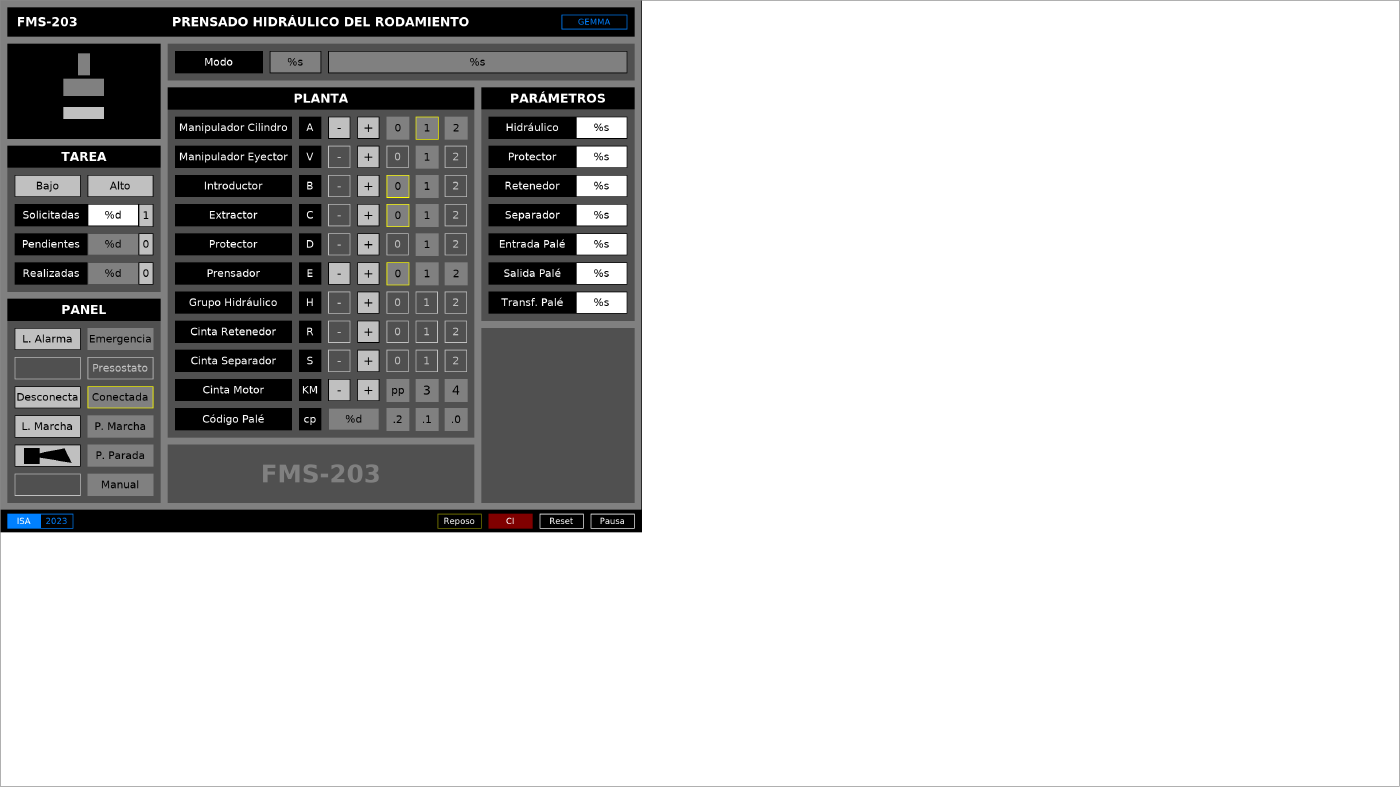
VISUALIZATION TC_VISU  // 1920x1080
    Rectangle (120,610 90x30)
    Rectangle (0,0 880x700)
    Rectangle (230,150 420x450)
    Rectangle (10,440 210x250)
    Rectangle (10,10 860x40), "PRENSADO HIDRÁULICO DEL RODAMIENTO"
    Rectangle (770,20 90x20), "GEMMA"
    Rectangle (10,60 210x130)
    Rectangle (230,120 420x30), "PLANTA"
    Rectangle (240,160 160x30), "Manipulador Cilindro"
    Rectangle (410,160 30x30), "A"
    Rectangle (450,160 30x30), "-"
    Rectangle (490,160 30x30), "+"
    Rectangle (530,160 30x30), "0"
    Rectangle (570,160 30x30), "1"
    Rectangle (610,160 30x30), "2"
    Rectangle (530,160 31x31), "0", colour toggle: MAIN.Estacion.ManipuladorDetras
        toggle MAIN.Estacion.ManipuladorDetras
    Rectangle (490,160 30x30), "+", colour toggle: MAIN.Estacion.ManipuladorAdelante
        toggle MAIN.Estacion.ManipuladorAdelante
    Rectangle (570,160 31x31), "1", colour toggle: MAIN.Estacion.ManipuladorMedio
        toggle MAIN.Estacion.ManipuladorMedio
    Rectangle (240,240 160x30), "Introductor"
    Rectangle (410,240 30x30), "B"
    Rectangle (10,410 210x30), "PANEL"
    Rectangle (20,450 90x30)
    Rectangle (0,700 880x30)
    Rectangle (55,705 45x20), "2023"
    Rectangle (10,705 45x20), "ISA"
    Rectangle (20,490 90x30)
    Rectangle (120,490 90x30), "Presostato"
    Rectangle (20,530 90x30)
    Rectangle (20,570 90x30)
    Rectangle (20,610 90x30)
    Rectangle (20,650 90x30)
    Rectangle (20,450 90x30), "L. Alarma", colour toggle: MAIN.Estacion.LamparaAlarma
        tap MAIN.Estacion.LamparaAlarma
    Rectangle (20,530 90x30), "Desconecta", colour toggle: MAIN.Estacion.DesconectaEstacion
        tap MAIN.Estacion.DesconectaEstacion
    Rectangle (20,570 90x30), "L. Marcha", colour toggle: MAIN.Estacion.LamparaMarcha
        tap MAIN.Estacion.LamparaMarcha
    Rectangle (20,610 90x30), colour toggle: MAIN.Estacion.AvisadorSonoro
        tap MAIN.Estacion.AvisadorSonoro
    Rectangle (120,450 90x30), colour toggle: MAIN.Estacion.PulsadorEmergencia
        toggle MAIN.Estacion.PulsadorEmergencia
    Rectangle (120,570 90x30)
    Rectangle (120,530 90x30)
    Rectangle (120,650 90x30)
    Rectangle (240,280 160x30), "Extractor"
    Rectangle (410,280 30x30), "C"
    Rectangle (240,320 160x30), "Protector"
    Rectangle (410,320 30x30), "D"
    Rectangle (240,360 160x30), "Prensador"
    Rectangle (410,360 30x30), "E"
    Rectangle (240,200 160x30), "Manipulador Eyector"
    Rectangle (410,200 30x30), "V"
    Rectangle (240,400 160x30), "Grupo Hidráulico"
    Rectangle (410,400 30x30), "H"
    Rectangle (240,440 160x30), "Cinta Retenedor"
    Rectangle (410,440 30x30), "R"
    Rectangle (240,480 160x30), "Cinta Separador"
    Rectangle (410,480 30x30), "S"
    Rectangle (240,520 160x30), "Cinta Motor"
    Rectangle (410,520 30x30), "KM"
    Rectangle (240,560 160x30), "Código Palé"
    Rectangle (410,560 30x30), "cp"
    Rectangle (230,610 420x80), "FMS-203"
    Rectangle (450,240 30x30), "-"
    Rectangle (490,240 30x30), "+"
    Rectangle (530,240 30x30), "0"
    Rectangle (570,240 30x30), "1"
    Rectangle (610,240 30x30), "2"
    Rectangle (530,240 31x31), "0", colour toggle: MAIN.Estacion.IntroductorDetras
        toggle MAIN.Estacion.IntroductorDetras
    Rectangle (490,240 30x30), "+", colour toggle: MAIN.Estacion.IntroductorAdelante
        toggle MAIN.Estacion.IntroductorAdelante
    Rectangle (570,240 31x31), "1", colour toggle: MAIN.Estacion.IntroductorDelante
        toggle MAIN.Estacion.IntroductorDelante
    Rectangle (450,280 30x30), "-"
    Rectangle (490,280 30x30), "+"
    Rectangle (530,280 30x30), "0"
    Rectangle (570,280 30x30), "1"
    Rectangle (610,280 30x30), "2"
    Rectangle (530,280 31x31), "0", colour toggle: MAIN.Estacion.ExtractorDetras
        toggle MAIN.Estacion.ExtractorDetras
    Rectangle (490,280 30x30), "+", colour toggle: MAIN.Estacion.ExtractorAdelante
        toggle MAIN.Estacion.ExtractorAdelante
    Rectangle (570,280 31x31), "1", colour toggle: MAIN.Estacion.ExtractorDelante
        toggle MAIN.Estacion.ExtractorDelante
    Rectangle (450,320 30x30), "-"
    Rectangle (490,320 30x30), "+"
    Rectangle (530,320 30x30), "0"
    Rectangle (570,320 30x30), "1"
    Rectangle (610,320 30x30), "2"
    Rectangle (490,320 30x30), "+", colour toggle: MAIN.Estacion.ProtectorBaja
        toggle MAIN.Estacion.ProtectorBaja
    Rectangle (570,320 31x31), "1", colour toggle: MAIN.Estacion.ProtectorAbajo
        toggle MAIN.Estacion.ProtectorAbajo
    Rectangle (450,360 30x30), "-"
    Rectangle (490,360 30x30), "+"
    Rectangle (530,360 30x30), "0"
    Rectangle (570,360 30x30), "1"
    Rectangle (610,360 30x30), "2"
    Rectangle (530,360 31x31), "0", colour toggle: MAIN.Estacion.PrensadorArriba
        toggle MAIN.Estacion.PrensadorArriba
    Rectangle (490,360 30x30), "+", colour toggle: MAIN.Estacion.PrensadorBaja
        toggle MAIN.Estacion.PrensadorBaja
    Rectangle (570,360 31x31), "1", colour toggle: MAIN.Estacion.PrensadorAbajoAlto
        toggle MAIN.Estacion.PrensadorAbajoAlto
    Rectangle (610,360 31x31), "2", colour toggle: MAIN.Estacion.PrensadorAbajoBajo
        toggle MAIN.Estacion.PrensadorAbajoBajo
    Rectangle (450,200 30x30), "-"
    Rectangle (450,360 30x30), "-", colour toggle: MAIN.Estacion.PrensadorSube
        toggle MAIN.Estacion.PrensadorSube
    Rectangle (490,200 30x30), "+"
    Rectangle (530,200 30x30), "0"
    Rectangle (570,200 30x30), "1"
    Rectangle (610,200 30x30), "2"
    Rectangle (490,200 30x30), "+", colour toggle: MAIN.Estacion.ManipuladorSucciona
        toggle MAIN.Estacion.ManipuladorSucciona
    Rectangle (570,200 31x31), "1", colour toggle: MAIN.Estacion.ManipuladorVacioObtenido
        toggle MAIN.Estacion.ManipuladorVacioObtenido
    Rectangle (450,400 30x30), "-"
    Rectangle (490,400 30x30), "+"
    Rectangle (530,400 30x30), "0"
    Rectangle (570,400 30x30), "1"
    Rectangle (610,400 30x30), "2"
    Rectangle (490,400 30x30), "+", colour toggle: MAIN.Estacion.HidraulicoActiva
        toggle MAIN.Estacion.HidraulicoActiva
    Rectangle (450,440 30x30), "-"
    Rectangle (490,440 30x30), "+"
    Rectangle (530,440 30x30), "0"
    Rectangle (570,440 30x30), "1"
    Rectangle (610,440 30x30), "2"
    Rectangle (490,440 30x30), "+", colour toggle: MAIN.Estacion.CintaRetenedorBaja
        toggle MAIN.Estacion.CintaRetenedorBaja
    Rectangle (450,480 30x30), "-"
    Rectangle (490,480 30x30), "+"
    Rectangle (530,480 30x30), "0"
    Rectangle (570,480 30x30), "1"
    Rectangle (610,480 30x30), "2"
    Rectangle (490,480 30x30), "+", colour toggle: MAIN.Estacion.CintaSeparadorSube
        toggle MAIN.Estacion.CintaSeparadorSube
    Rectangle (450,520 30x30), "-"
    Rectangle (450,520 30x30), "-", colour toggle: MAIN.Estacion.CintaMotorInvierte
        toggle MAIN.Estacion.CintaMotorInvierte
    Rectangle (490,520 30x30), "+"
    Rectangle (530,520 30x30), "0"
    Rectangle (570,520 30x30), "1"
    Rectangle (610,520 30x30), "2"
    Rectangle (530,520 31x31), "pp", colour toggle: MAIN.Estacion.PalePresencia
        toggle MAIN.Estacion.PalePresencia
    Rectangle (490,520 30x30), "+", colour toggle: MAIN.Estacion.CintaMotorActiva
        toggle MAIN.Estacion.CintaMotorActiva
    Rectangle (570,520 31x31), "3", colour toggle: MAIN.Estacion.CintaMotorActiva AND MAIN.Estacion.CintaMotorInvierte
    Rectangle (450,560 30x30), "-"
    Rectangle (490,560 30x30), "+"
    Rectangle (530,560 30x30), "0"
    Rectangle (570,560 30x30), "1"
    Rectangle (610,560 30x30), "2"
    Rectangle (530,560 31x31), ".2", colour toggle: MAIN.Estacion.PaleCodigoBit2
        toggle MAIN.Estacion.PaleCodigoBit2
    Rectangle (610,560 31x31), ".0", colour toggle: MAIN.Estacion.PaleCodigoBit0
        toggle MAIN.Estacion.PaleCodigoBit0
    Rectangle (570,560 31x31), ".1", colour toggle: MAIN.Estacion.PaleCodigoBit1
        toggle MAIN.Estacion.PaleCodigoBit1
    Rectangle (450,560 70x30), "%d", text variable: MAIN.Estacion.PaleCodigo
    Rectangle (610,520 31x31), "4", colour toggle: MAIN.Estacion.CintaMotorActiva AND NOT MAIN.Estacion.CintaMotorInvierte
    Rectangle (120,530 90x30), "Conectada", colour toggle: MAIN.Estacion.EstacionConectada
        toggle MAIN.Estacion.EstacionConectada
    Rectangle (120,570 90x30), "P. Marcha", colour toggle: MAIN.Estacion.PulsadorMarcha
        tap MAIN.Estacion.PulsadorMarcha
    Rectangle (120,450 90x30), "Emergencia", colour toggle: MAIN.Estacion.PulsadorEmergencia
        toggle MAIN.Estacion.PulsadorEmergencia
    Rectangle (120,650 90x30), "Manual", colour toggle: MAIN.Estacion.SelectorManual
        toggle MAIN.Estacion.SelectorManual
    Rectangle (120,610 90x30)
    Rectangle (120,610 90x30), "P. Parada", colour toggle: MAIN.Estacion.PulsadorParada
        tap MAIN.Estacion.PulsadorParada p1329445385=TRUE
    Group (56,71 119x109)
        Group (0,0 117x107)
            Polygon (119,109)
            Polygon (0,109)
            Polyline (40,94)
            Polyline (30,86)
            Polyline (30,76)
            Polyline (30,66)
            Polyline (40,54)
            Polyline (119,104)
            Polyline (119,94)
            Polyline (119,84)
            Polyline (119,74)
            Polyline (119,54)
            Rectangle (29,35 59x27)
            Rectangle (49,0 20x34)
            Rectangle (49,22 20x12)
            Rectangle (29,63 59x10)
            Polyline (40,104)
            Polyline (118,64)
            Rectangle (29,74 59x20)
        Polygon (119,109)
        Polygon (0,109)
        Polyline (40,94)
        Polyline (30,86)
        Polyline (30,76)
        Polyline (30,66)
        Polyline (40,54)
        Polyline (119,104)
        Polyline (119,94)
        Polyline (119,84)
        Polyline (119,74)
        Polyline (119,54)
        Rectangle (29,35 59x27)
        Rectangle (49,0 20x34)
        Rectangle (29,63 59x10)
        Polyline (40,104)
        Polyline (118,64)
        Rectangle (29,74 59x20)
    Rectangle (610,160 31x31), "2", colour toggle: MAIN.Estacion.ManipuladorDelante
        toggle MAIN.Estacion.ManipuladorDelante
    Group (33,615 65x21)
        tap MAIN.Estacion.AvisadorSonoro
        Rectangle (0,0 21x21)
        Polygon (5,10) (55,0) (55,0) (65,20) (5,10)
    Rectangle (660,120 210x30), "PARÁMETROS"
    Rectangle (660,150 210x290)
    Rectangle (670,160 120x30), "Hidráulico"
    Rectangle (790,160 70x30), "%s", text variable: MAIN.Estacion.TpoPrensaHidraulico
        OnMouseClick: write the text variable via Default
    Rectangle (670,200 120x30), "Protector"
    Rectangle (670,240 120x30), "Retenedor"
    Rectangle (670,280 120x30), "Separador"
    Rectangle (670,320 120x30), "Entrada Palé"
    Rectangle (670,360 120x30), "Salida Palé"
    Rectangle (670,400 120x30), "Transf. Palé"
    Rectangle (790,200 70x30), "%s", text variable: MAIN.Estacion.TpoPrensaProtector
        OnMouseClick: write the text variable via Default
    Rectangle (790,240 70x30), "%s", text variable: MAIN.Estacion.TpoCintaRetenedor
        OnMouseClick: write the text variable via Default
    Rectangle (790,280 70x30), "%s", text variable: MAIN.Estacion.TpoCintaSeparador
        OnMouseClick: write the text variable via Default
    Rectangle (790,320 70x30), "%s", text variable: MAIN.Estacion.TpoPaleEntrada
        OnMouseClick: write the text variable via Default
    Rectangle (790,360 70x30), "%s", text variable: MAIN.Estacion.TpoPaleSalida
        OnMouseClick: write the text variable via Default
    Rectangle (790,400 70x30), "%s", text variable: MAIN.Estacion.TpoPaleTransferencia
        OnMouseClick: write the text variable via Default
    Rectangle (10,200 210x30), "TAREA"
    Rectangle (10,230 210x170)
    Rectangle (120,240 90x30), "Alto", colour toggle: NOT MAIN.Estacion.RodamientoBajo
        OnMouseClick: execute { MAIN.Estacion.RodamientoBajo := FALSE; }
    Rectangle (20,280 100x30), "Solicitadas"
    Rectangle (120,280 70x30), "%d", text variable: MAIN.Estacion.UnidadesSolicitadas
        OnMouseClick: write the text variable via Default, min 1
    Rectangle (20,320 100x30), "Pendientes"
    Rectangle (120,320 70x30), "%d", text variable: MAIN.Estacion.UnidadesPendientes
        OnMouseClick: write the text variable via Default
    Rectangle (20,360 100x30), "Realizadas"
    Rectangle (120,360 70x30), "%d", text variable: MAIN.Estacion.UnidadesRealizadas
        OnMouseClick: write the text variable via Default
    Rectangle (20,240 90x30), "Bajo", colour toggle: MAIN.Estacion.RodamientoBajo
        OnMouseClick: execute { MAIN.Estacion.RodamientoBajo := TRUE; }
    Rectangle (660,450 210x240)
    Rectangle (450,160 30x30), "-", colour toggle: MAIN.Estacion.ManipuladorAtras
        toggle MAIN.Estacion.ManipuladorAtras
    RoundedRectangle (670,705 60x20), "CI"
    RoundedRectangle (670,705 60x20), "CI", colour toggle: MAIN.Estacion.CondicionInicial, invisible if: NOT MAIN.Estacion.Coordinador.Ready
    RoundedRectangle (740,705 60x20), "Reset", colour toggle: MAIN.Estacion.EstadoReinicia, invisible if: NOT MAIN.FMS203.Reposo
        tap MAIN.Estacion.EstadoReinicia
    RoundedRectangle (600,705 60x20), "Reposo", colour toggle: MAIN.Estacion.Coordinador.Ready
    Rectangle (190,280 20x31), "1"
        OnMouseClick: execute { MAIN.Estacion.UnidadesSolicitadas := 1 }
    Rectangle (190,320 20x30), "0"
        OnMouseClick: execute { MAIN.Estacion.UnidadesPendientes := 0 }
    Rectangle (190,360 20x30), "0"
        OnMouseClick: execute { MAIN.Estacion.UnidadesRealizadas := 0 }
    RoundedRectangle (810,705 60x20), "Pausa", colour toggle: MAIN.Estacion.EstadoPausa, invisible if: NOT MAIN.FMS203.Reposo
        toggle MAIN.Estacion.EstadoPausa
    Rectangle (230,60 640x50)
    Rectangle (240,70 120x30), "Modo"
    Rectangle (370,70 70x30), "%s", text variable: MAIN.Estacion.Director.Modo
    Rectangle (450,70 410x30), "%s", text list: 'ModoDescripcion', text index: MAIN.Estacion.Director.Modo
    Rectangle (20,15 120x30), "FMS-203"
END_VISUALIZATION

(* stored: Version 1.1.0.1, ProductVersion 3.1.4024.12
   Visu TC_VISU: Id {25fd3f38-3886-4040-8a7c-9b698307486c} *)
